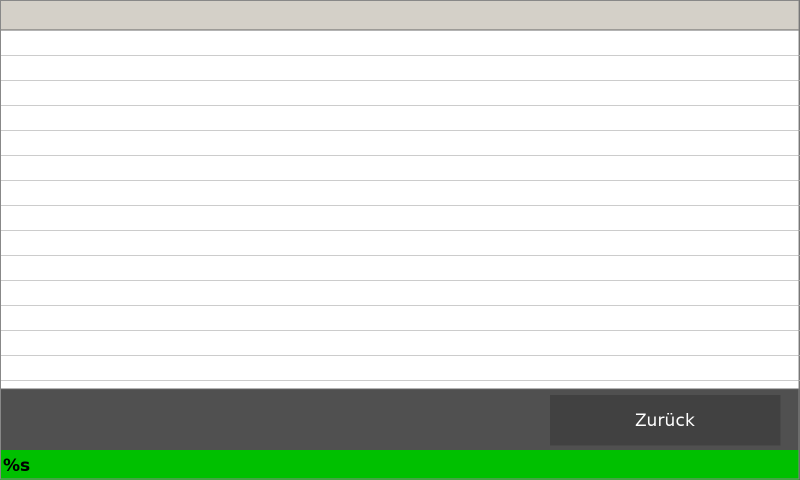
VISUALIZATION EventLogger  // 800x480
    Table (0,0 800x389), data array: EventLogger.aLoggedEvents
        p3854506369: EventLogger.aLoggedEvents[INDEX].sSeverity
        p1892666644: EventLogger.aLoggedEvents[INDEX].sStatus
        p338671338: EventLogger.aLoggedEvents[INDEX].sTimestamp
        p2170511999: EventLogger.aLoggedEvents[INDEX].sText
        p3723444502: EventLogger.aLoggedEvents[INDEX].nEventId
        p1218418051: EventLogger.aLoggedEvents[INDEX].bPinned
        p1755163831: Zeit
        p4092479075: Fehlermeldung
    Rectangle (550,395 230x50), "Zurück"
        OnMouseClick: change screen: Previous Zyklusbetrieb
    Rectangle (0,450 799x30), "%s", text variable: MAIN.HMI.sStatus, colour variable: MAIN.HMI.nColorInfoBalken
        p3450524324: MAIN.HMI.nColorInfoBalken
END_VISUALIZATION

(* stored: Version 1.1.0.1, ProductVersion 3.1.4024.12
   Visu EventLogger: Id {1aa99805-375e-4624-add5-94d9fdb9a033} *)
